FUNCTION Convert_REAL_TO_LINT : BOOL
VAR_INPUT
	in : REAL;
	out : REFERENCE TO LINT;
END_VAR
VAR
	converted : LINT;
END_VAR

converted := REAL_TO_LINT(in);

IF (LINT_TO_REAL(converted) <> in) THEN
	RETURN;
END_IF

out := converted;
Convert_REAL_TO_LINT := TRUE;

END_FUNCTION

(* stored: Version 1.1.0.1, ProductVersion 3.1.4024.12
   POU Convert_REAL_TO_LINT: Id {86571434-7f48-40f7-bd84-fea333bd2d4a}, SpecialFunc None *)
